{attribute 'qualified_only'}
{attribute 'strict'}
TYPE ePositionType :
(
	POSITION_ABS := 0,
	POSITION_REL := 1
);
END_TYPE

(* stored: Version 1.1.0.1, ProductVersion 3.1.4022.10
   DUT ePositionType: Id {55de27bb-a4c8-4ace-84de-fb78476b5140} *)
